Staubli VAL3: N17_AproTirarPuntes.pgx

program N17_AproTirarPuntes()
  local pointRx l_pAproTirarPuntes
begin

  // Anar a l'aproximació del punt de tirar puntes
  l_pAproTirarPuntes=pTirarPuntes
  l_pAproTirarPuntes.trsf.x=l_pAproTirarPuntes.trsf.x+nXOffset
  l_pAproTirarPuntes.trsf.y=l_pAproTirarPuntes.trsf.y+nYOffset
  l_pAproTirarPuntes.trsf.z=l_pAproTirarPuntes.trsf.z+nZOffset

  if nZApro>0
    l_pAproTirarPuntes.trsf.z=l_pAproTirarPuntes.trsf.z+nZApro
  else
    l_pAproTirarPuntes.trsf.z=l_pAproTirarPuntes.trsf.z+50
  endIf

  movel(l_pAproTirarPuntes,tToolActiva,mLent)
  waitEndMove()

  bTaskDone=true
end
